TYPE ST_Pompe_Prio :
STRUCT
PmpID				:INT;
Dispox				:BOOL;
PmpPrioNumero		:INT;
Allume				:BOOL;


	

END_STRUCT
END_TYPE

(* stored: Version 1.1.0.1, ProductVersion 3.1.4024.12
   DUT ST_Pompe_Prio: Id {32e4fba3-1df3-413f-a2ea-384ea88fd9cb} *)
